Staubli VAL3: onF1Event.pgx

program onF1Event(string x_sItem (dimensions=1), bool& x_bSave[] (dimensions=1))
  local bool l_bChange
  local bool l_bStatus
begin
  // look if the bButton is enable
  if bButton[0]
    if sMode=="OUT"
      // OUTPUT
      call out:isEnable(l_bStatus,x_sItem)
      call out:setEnable(!l_bStatus,x_sItem)
      logMsg("[KERNEL] INTERFACE:Change the active status of: "+x_sItem)
    elseIf sMode=="IN"
      // INPUT
      call in:isEnable(l_bStatus,x_sItem)
      call in:setEnable(!l_bStatus,x_sItem)
      logMsg("[KERNEL] INTERFACE:Change the active status of: "+x_sItem)
    endIf
    // save it
    x_bSave=true
  endIf
end
